TYPE CanOverEthercatConfig :
STRUCT
	CoeSerialComSettings : CoeSerialComSettings;
END_STRUCT
END_TYPE

(* stored: Version 1.1.0.1, ProductVersion 3.1.4024.3
   DUT CanOverEthercatConfig: Id {9daa58a8-526a-4fc0-9fca-a815424e3d14} *)
